{attribute 'GeneratedUsingTerminal: EK1100-0000-0018'}
{attribute addProperty BoxType "EK1100-0000-0018"}
{attribute addProperty Id "Beckhoff_CUxxxxEK1122Beckhoff_CUxxxxEK1122_1D92BB5F94"}
{attribute addProperty CRC "3784165595"}
{attribute addProperty Size "94"}
TYPE Beckhoff_CUxxxx_E18DC8DB EXTENDS EK1100_1FC0878B :
STRUCT
	{attribute addProperty Name "Beckhoff_CUxxxxEK1122"}
	{attribute addProperty PreviousPort "Beckhoff CUxxxx : B"}
	Beckhoff_CUxxxxEK1122 : Beckhoff_CUxxxxEK1122_1D92BB5F;
END_STRUCT
END_TYPE

(* stored: Version 1.2.0.0, ProductVersion 3.1.4024.9
   DUT Beckhoff_CUxxxx_E18DC8DB: Id {91996b70-6b17-46a5-b6c3-ae34b546f24c} *)
